# EPICS StreamDevice protocol: protocols/capstat.proto
Terminator = LF;
ExtraInput = Ignore;

getBusy {
        in "BUSY=%d";
}
